PROGRAM S12_PreLine
VAR
END_VAR

END_PROGRAM

(* stored: Version 1.1.0.1, ProductVersion 3.1.4024.9
   POU S12_PreLine: Id {ebde0494-312e-4ed1-9c94-463f75f332eb}, SpecialFunc None *)
